FUNCTION alg_M_Distributing_a_Dstartled : BOOL
VAR_INPUT
	state: STATE;
END_VAR

alg_M_Distributing_a_Dstartled := (((state.dvar_M_Distributing) <> (elit_wait_start)) AND ((state.dvar_M_Distributing) <> (elit_init2))) AND ((state.dvar_M_Distributing) <> (elit_stop));

END_FUNCTION

(* stored: Version 1.1.0.1, ProductVersion 3.1.4022.18
   POU alg_M_Distributing_a_Dstartled: Id {83734109-358d-4081-9f24-df7354195d68}, SpecialFunc None *)
